Staubli VAL3: robotGet.pgx

public program robotGet(point pPosition, trsf trTrans, tool tTool, mdesc mApproach, mdesc mTarget)
  local point pAppro
begin
  // Picks a part
  //
  // copyright (c) 2015-2018 victortorreslopez
  //
  // GNU General Public License
  //
  // Parameters
  // - pPosition: target position
  // - trTrans: approach transform to target position
  // - tTool: current tool
  // - mApproach: movement descriptor to "approach" point
  // - mTarget: movement descriptor to "target" position
  //
  // Local variables
  // - pAppro: approach point to target position
  //
  // References
  // - "2005-27 Example Application". Staubli. 2005
  //
  // Version history
  // ---------------
  // 2.0, 2020/02/15, VTL: renames all parameters
  // 1.1, 2018/09/27, VTL: adds "ma"
  // 1.0, 2018/09/27, VTL: renames "m" by "mt"
  // 0.0, 2015/01/14, VTL: alfa release

  pAppro = appro(pPosition, trTrans)
  movej(pAppro, tTool, mApproach)
  movel(pPosition, tTool, mTarget)
  close(tTool)
  movel(pAppro, tTool, mTarget)
end
